FUNCTION Convert_BYTE_TO_LINT : BOOL
VAR_INPUT
	in : BYTE;
	out : REFERENCE TO LINT;
END_VAR
VAR
	converted : LINT;
END_VAR

converted := BYTE_TO_LINT(in);

IF (LINT_TO_BYTE(converted) <> in) THEN
	RETURN;
END_IF

out := converted;
Convert_BYTE_TO_LINT := TRUE;

END_FUNCTION

(* stored: Version 1.1.0.1, ProductVersion 3.1.4024.12
   POU Convert_BYTE_TO_LINT: Id {e5e70ecc-4f28-4f02-8d93-d6262f2653a8}, SpecialFunc None *)
